INTERFACE I_Collection EXTENDS I_Enumerator

METHOD AddItem
VAR_INPUT
	Item : I_Base;
END_VAR
END_METHOD

METHOD Clear
VAR_INPUT
END_VAR
END_METHOD

{attribute 'monitoring' := 'call'}
PROPERTY Count : UDINT
GET
END_GET
END_PROPERTY

{attribute 'monitoring' := 'call'}
PROPERTY IsEmpty : BOOL
GET
END_GET
END_PROPERTY

METHOD RemoveItem
VAR_INPUT
	Item : I_Base;
END_VAR
END_METHOD

END_INTERFACE

(* stored: Version 1.1.0.1, ProductVersion 3.1.4026.18
   Itf I_Collection: Id {c757555d-4a1d-49bf-8710-866778da8742}
   Method AddItem: Id {2d6767a3-2140-4c48-ba5d-63344ac016a3}
   Method Clear: Id {79dae6dc-2d10-437d-b5eb-68284dbb1438}
   Property Count: Id {4e1decf6-5bbb-40a6-a343-dc1340df0ca0}
   Get Get: Id {5cfc5a90-3f7e-45f2-88fc-a0096cdd3872}
   Property IsEmpty: Id {fc97bf38-a655-4efe-9740-40b141064c1b}
   Get Get: Id {87db1896-9e25-4dbd-a403-90045b330513}
   Method RemoveItem: Id {89e998f2-649f-4e35-9265-7b42ca0dddf7} *)
